TYPE ST_BhFMStatus :
STRUCT
	
uiFlowPercentageRaw	:	UINT;
	rFlowPercentage	: REAL;
	rFlow	:	REAL;
	xOoR	:	BOOL; // Out of range above
xFlowValid	:	BOOL;
	sReply	:	STRING;
	iState	:	INT;

END_STRUCT
END_TYPE

(* stored: Version 1.1.0.1, ProductVersion 3.1.4020.12
   DUT ST_BhFMStatus: Id {956ac3ba-fa11-4079-a7f0-2e4d7c89266b} *)
